(* Logix 5000 project; controller Proceso_Corte_de_bambu Emulate 5570 rev 32.11; software revision 32.00 *)

TASK MainTask (continuous, watchdog 500 ms) : MainProgram

MODULES
   Local : Emulate 5570 (ICP 4, rev 32.11)
      INPUTS_OUTPUTS : vendor 1 type 0 code 15 (ICP 3, rev 1.1, Output RPI 150 ms)
END_MODULES

PROGRAM MainProgram   (* main routine MainRoutine *)
VAR
   Banda : ALIAS FOR Local:3:O.Data[0].0;
   Banda_time0 : TIMER := (PRE := 2000);
   Banda_time1 : TIMER := (PRE := 500);
   habilitado : BOOL;
   oneshot : BOOL;
   pos_cil_act : REAL;
   pos_cil_sig : REAL;
   pos_suj_act : REAL;
   pos_suj_sig : REAL;
   sensor_active : BOOL;
   sensor_actived : BOOL;
   sierra_ac : ALIAS FOR Local:3:O.Data[0].2;
   sierra_cnt : COUNTER := (PRE := 1);
   sierra_M : ALIAS FOR Local:3:O.Data[0].4;
   sierra_ret : ALIAS FOR Local:3:O.Data[0].3;
   sierra_up : ALIAS FOR Local:3:I.Data[1].2;
   START : ALIAS FOR Local:3:I.Data[1].0;
   Step_000 : SFC_STEP := (Status := 16#0020_0000, PauseTimer := 1);
   STOP : ALIAS FOR Local:3:I.Data[1].1;
   suj_pos_ini : ALIAS FOR Local:3:I.Data[1].3;
   suj_time : TIMER := (PRE := 2000);
   sujecion_ac : ALIAS FOR Local:3:O.Data[0].1;
   sujecion_ret : ALIAS FOR Local:3:O.Data[0].5;
   Tran_000 : BOOL;
END_VAR

ROUTINE MainRoutine   (* ladder *)
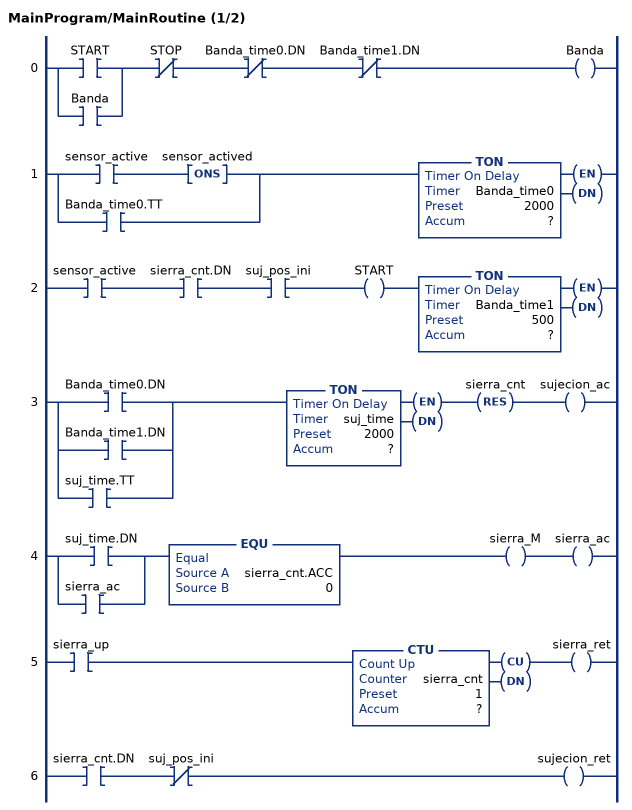
   0: [XIC(START) ,XIC(Banda) ]XIO(STOP)XIO(Banda_time0.DN)XIO(Banda_time1.DN)OTE(Banda);
   1: [XIC(sensor_active) ONS(sensor_actived) ,XIC(Banda_time0.TT) ]TON(Banda_time0,?,?);
   2: XIC(sensor_active)XIC(sierra_cnt.DN)XIC(suj_pos_ini)OTE(START)TON(Banda_time1,?,?);
   3: [XIC(Banda_time0.DN) ,XIC(Banda_time1.DN) ,XIC(suj_time.TT) ]TON(suj_time,?,?)RES(sierra_cnt)OTE(sujecion_ac);
   4: [XIC(suj_time.DN) ,XIC(sierra_ac) ]EQU(sierra_cnt.ACC,0)OTE(sierra_M)OTE(sierra_ac);
   5: XIC(sierra_up)CTU(sierra_cnt,?,?)OTE(sierra_ret);
   6: XIC(sierra_cnt.DN)XIO(suj_pos_ini)OTE(sujecion_ret);
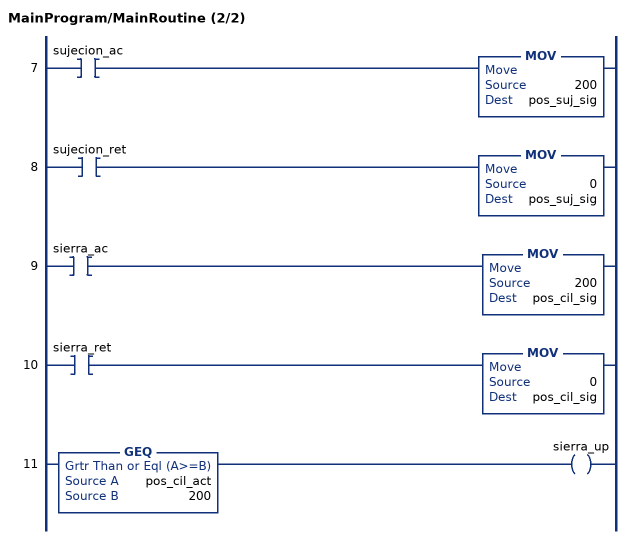
   7: XIC(sujecion_ac)MOV(200,pos_suj_sig);
   8: XIC(sujecion_ret)MOV(0,pos_suj_sig);
   9: XIC(sierra_ac)MOV(200,pos_cil_sig);
   10: XIC(sierra_ret)MOV(0,pos_cil_sig);
   11: GEQ(pos_cil_act,200)OTE(sierra_up);
END_ROUTINE
END_PROGRAM
